FUNCTION_BLOCK FB_ExecuteGcode
VAR_INPUT
	sPrgName: STRING(255);
	execute: BOOL;
	in_stNciToPlc: NCTOPLC_NCICHANNEL_REF;
	reset: bool := FALSE;
END_VAR
VAR_OUTPUT
	done: BOOL;
END_VAR
VAR
	state: INT := 0;
	nInterpreterState: UDINT;
	
	fbLoadGCode: ItpLoadProgEx;
	fbStartGCode: ItpStartStopEx;
	
END_VAR

CASE state OF
	0:
	IF execute = TRUE THEN
		done:=FALSE;
		state:= 10;
	END_IF
	
	10:// laad g-code
	fbLoadGCode(
		sNciToPlc:=in_stNciToPlc, 
		bExecute:=TRUE, 
		sPrg:= sPrgName, 
		nLength:= INT_TO_UDINT(LEN(sPrgName)) );
	IF NOT fbLoadGCode.bBusy THEN
		IF NOT fbLoadGCode.bErr THEN
			State	:= 20;				
		END_IF
		fbLoadGCode(sNciToPlc:=in_stNciToPlc, bExecute:=FALSE); 
	END_IF 
	
	20:// check status NCI
	fbLoadGCode(
		sNciToPlc:=in_stNciToPlc, 
		bExecute:=FALSE);
	nInterpreterState	:= ItpGetStateInterpreter(sNciToPlc:=in_stNciToPlc);
	IF nInterpreterState = Tc2_NCI.NCI_INTERPRETER_READY THEN // als de interpreter klaar is kan het programma verder
			State	:= 30;	
	END_IF
	
	30: // start g-code
	fbStartGCode(
		bStart:=TRUE, 
		bStop:=FALSE, 
		tTimeOut:= , 
		sNciToPlc:= in_stNciToPlc, 
		bBusy=> , 
		bErr=> , 
		nErrId=> );
	IF NOT fbStartGCode.bBusy THEN
		IF NOT fbStartGCode.bErr THEN
			State	:= 40;			
		END_IF
		fbStartGCode( bStart:= FALSE, sNciToPlc:= in_stNciToPlc); 
	END_IF
	
	40: // g-code is gestart
	fbStartGCode( bStart:= FALSE, sNciToPlc:= in_stNciToPlc);
	done := TRUE;
	state := 50;
	
	50:
	IF reset = TRUE THEN
		state := 0;
	END_IF
	
END_CASE

END_FUNCTION_BLOCK

(* stored: Version 1.1.0.1, ProductVersion 3.1.4024.9
   POU FB_ExecuteGcode: Id {2069b1af-391a-4a29-945a-fe64923ed0d3}, SpecialFunc None *)
